(* IEC 61131-3 sources: AXOpen/src/components.cognex.vision/app/src/Documentation, 6 files *)

(* ---- Component_1.st ---- *)
USING AXOpen.Core;

NAMESPACE AXOpen.Components.Cognex.Vision

    {S7.extern=ReadWrite}
    CLASS Component_1 EXTENDS AXOpen.Core.AxoObject
        //<ComponentDeclaration>
        VAR PUBLIC
            Insight_7600 : AXOpen.Components.Cognex.Vision.v_6_0_0_0.AxoInsight;
        END_VAR
        //</ComponentDeclaration>

        //<InitializationArgumentsDeclaration>
        VAR PUBLIC
            {#ix-set:AttributeName = "<#Activate manual control#>"}
            ActivateManualControl : BOOL;
        END_VAR
        //</InitializationArgumentsDeclaration>

        METHOD PUBLIC OVERRIDE Run
            VAR_INPUT
                parent : IAxoObject;
            END_VAR

            SUPER.Run(parent);

            IF ActivateManualControl THEN
                //<InsightManualControl>
                Insight_7600.ActivateManualControl();
                //</InsightManualControl>
            END_IF;

            //<Initialization>
            Insight_7600.Run(parent := THIS, hwID :=  HwIdentifiers#is7600_HwID);
            //</Initialization>
            THIS.UseInSequencer();
        END_METHOD

        //<Usage>
        VAR PUBLIC
            Sequencer : AxoSequencer;
            Steps : ARRAY[0..10] OF AXOpen.Core.AxoStep;
        END_VAR

        VAR PRIVATE
            _InspectionResults  :   AXOpen.Components.Cognex.Vision.v_6_0_0_0.AxoInsight_ResultData;
        END_VAR

        METHOD PRIVATE UseInSequencer
            IF Sequencer.GetContext().OpenCycleCount() <= ULINT#10 THEN
                Sequencer.SequenceMode := eAxoSequenceMode#RunOnce;
            END_IF;

            Sequencer.Run(THIS);
            Sequencer.Open();

            IF(Steps[0].Execute(Sequencer, 'Restore')) THEN
                Insight_7600.Restore();
                Sequencer.MoveNext();
            END_IF;

            IF(Steps[1].Execute(Sequencer, 'Change job: 1_test01.job')) THEN
                IF(Insight_7600.ChangeJob('1_test01.job').IsDone()) THEN
                    Sequencer.MoveNext();
                END_IF;
            END_IF;

            IF(Steps[2].Execute(Sequencer, 'Trigger')) THEN
                IF(Insight_7600.Trigger().IsDone()) THEN
                    Sequencer.MoveNext();
                END_IF;
            END_IF;

            IF(Steps[3].Execute(Sequencer, 'Evaluate inspection results')) THEN
                _InspectionResults := Insight_7600.InspectionResults;
                Sequencer.MoveNext();
            END_IF;

            IF(Steps[4].Execute(Sequencer, 'Clear inspaction results')) THEN
                IF(Insight_7600.ClearInspectionResults().IsDone()) THEN
                    Sequencer.MoveNext();
                END_IF;
            END_IF;

            IF(Steps[5].Execute(Sequencer, 'Soft event')) THEN
                IF(Insight_7600.SoftEvent(UINT#5).IsDone()) THEN
                    Sequencer.MoveNext();
                END_IF;
            END_IF;

            IF(Steps[6].Execute(Sequencer, 'Restore')) THEN
                Insight_7600.Restore();
                Sequencer.CompleteSequence();
            END_IF;

        END_METHOD

        //</Usage>

    END_CLASS
END_NAMESPACE

(* ---- Component_2.st ---- *)
USING AXOpen.Core;

NAMESPACE AXOpen.Components.Cognex.Vision.v_6_0_0_0

    {S7.extern=ReadWrite}
    CLASS Component_2 EXTENDS AXOpen.Core.AxoObject
        //<ComponentDeclaration>
        VAR PUBLIC
            Dataman_280 : AXOpen.Components.Cognex.Vision.v_6_0_0_0.AxoDataman;
        END_VAR
        //</ComponentDeclaration>

        //<InitializationArgumentsDeclaration>
        VAR PUBLIC
            {#ix-set:AttributeName = "<#Activate manual control#>"}
            ActivateManualControl : BOOL;
        END_VAR
        //</InitializationArgumentsDeclaration>

        METHOD PUBLIC OVERRIDE Run
            VAR_INPUT
                parent : IAxoObject;
            END_VAR

            SUPER.Run(parent);

            IF ActivateManualControl THEN
                //<DatamanManualControl>
                Dataman_280.ActivateManualControl();
                //</DatamanManualControl>
            END_IF;

            //<Initialization>
            Dataman_280.Run(parent  :=  THIS, hwID :=  HwIdentifiers#dm_280_HwID);
            //</Initialization>

            THIS.UseInSequencer();
        END_METHOD

        //<Usage>
        VAR PUBLIC
            Sequencer : AxoSequencer;
            Steps : ARRAY[0..10] OF AXOpen.Core.AxoStep;
        END_VAR

        VAR PRIVATE
            _ResultData  :   AXOpen.Components.Cognex.Vision.v_6_0_0_0.AxoDataman_ResultData;
        END_VAR

        METHOD PRIVATE UseInSequencer
            IF Sequencer.GetContext().OpenCycleCount() <= ULINT#10 THEN
                Sequencer.SequenceMode := eAxoSequenceMode#RunOnce;
            END_IF;

            Sequencer.Run(THIS);
            Sequencer.Open();

            IF(Steps[0].Execute(Sequencer, 'Restore')) THEN
                Dataman_280.Restore();
                Sequencer.MoveNext();
            END_IF;

            IF(Steps[1].Execute(Sequencer, 'Clear result data')) THEN
                IF(Dataman_280.ClearResultData().IsDone()) THEN
                    Sequencer.MoveNext();
                END_IF;
            END_IF;

            IF(Steps[2].Execute(Sequencer, 'Read data')) THEN
                IF(Dataman_280.Read().IsDone()) THEN
                    Sequencer.MoveNext();
                END_IF;
            END_IF;

            IF(Steps[3].Execute(Sequencer, 'Evaluate data')) THEN
                _ResultData := Dataman_280.ResultData;
                Sequencer.MoveNext();
            END_IF;

            IF(Steps[4].Execute(Sequencer, 'Restore')) THEN
                Dataman_280.Restore();
                Sequencer.CompleteSequence();
            END_IF;

        END_METHOD

        //</Usage>
    END_CLASS
END_NAMESPACE

(* ---- Component_3.st ---- *)
USING AXOpen.Core;

NAMESPACE AXOpen.Components.Cognex.Vision

    {S7.extern=ReadWrite}
    CLASS Component_3 EXTENDS AXOpen.Core.AxoObject
        //<ComponentDeclaration>
        VAR PUBLIC
            Dataman_300 : AXOpen.Components.Cognex.Vision.v_6_0_0_0.AxoDataman;
        END_VAR
        //</ComponentDeclaration>

        //<InitializationArgumentsDeclaration>
        VAR PUBLIC
            {#ix-set:AttributeName = "<#Activate manual control#>"}
            ActivateManualControl : BOOL;
        END_VAR
        //</InitializationArgumentsDeclaration>

        METHOD PUBLIC OVERRIDE Run
            VAR_INPUT
                parent : IAxoObject;
            END_VAR

            SUPER.Run(parent);

            IF ActivateManualControl THEN
                //<DatamanManualControl>
                Dataman_300.ActivateManualControl();
                //</DatamanManualControl>
            END_IF;

            //<Initialization>
            Dataman_300.Run(parent := THIS, hwID :=  HwIdentifiers#dm_300_HwID);
            //</Initialization>

        THIS.UseInSequencer();
        END_METHOD

        //<Usage>
        VAR PUBLIC
            Sequencer : AxoSequencer;
            Steps : ARRAY[0..10] OF AXOpen.Core.AxoStep;
        END_VAR

        VAR PRIVATE
            _ResultData  :   AXOpen.Components.Cognex.Vision.v_6_0_0_0.AxoDataman_ResultData;
        END_VAR

        METHOD PRIVATE UseInSequencer
            IF Sequencer.GetContext().OpenCycleCount() <= ULINT#10 THEN
                Sequencer.SequenceMode := eAxoSequenceMode#RunOnce;
            END_IF;

            Sequencer.Run(THIS);
            Sequencer.Open();

            IF(Steps[0].Execute(Sequencer, 'Restore')) THEN
                Dataman_300.Restore();
                Sequencer.MoveNext();
            END_IF;

            IF(Steps[1].Execute(Sequencer, 'Clear result data')) THEN
                IF(Dataman_300.ClearResultData().IsDone()) THEN
                    Sequencer.MoveNext();
                END_IF;
            END_IF;

            IF(Steps[2].Execute(Sequencer, 'Read data')) THEN
                IF(Dataman_300.Read().IsDone()) THEN
                    Sequencer.MoveNext();
                END_IF;
            END_IF;

            IF(Steps[3].Execute(Sequencer, 'Evaluate data')) THEN
                _ResultData := Dataman_300.ResultData;
                Sequencer.MoveNext();
            END_IF;

            IF(Steps[4].Execute(Sequencer, 'Restore')) THEN
                Dataman_300.Restore();
                Sequencer.CompleteSequence();
            END_IF;

        END_METHOD

        //</Usage>
    END_CLASS
END_NAMESPACE

(* ---- Component_4.st ---- *)
USING AXOpen.Core;

NAMESPACE AXOpen.Components.Cognex.Vision

    {S7.extern=ReadWrite}
    CLASS Component_4 EXTENDS AXOpen.Core.AxoObject
        //<ComponentDeclaration>
        VAR PUBLIC
            Insight_2800 : AXOpen.Components.Cognex.Vision.v_24_0_0.AxoInsight;
        END_VAR
        //</ComponentDeclaration>

        //<InitializationArgumentsDeclaration>
        VAR PUBLIC
            {#ix-set:AttributeName = "<#Activate manual control#>"}
            ActivateManualControl : BOOL;
        END_VAR
        //</InitializationArgumentsDeclaration>

        METHOD PUBLIC OVERRIDE Run
            VAR_INPUT
                inParent : IAxoObject;
            END_VAR

            SUPER.Run(inParent);

            IF ActivateManualControl THEN
                //<InsightManualControl>
                Insight_2800.ActivateManualControl();
                //</InsightManualControl>
            END_IF;

            //<Initialization>
            Insight_2800.Run(parent := THIS, hwID := HwIdentifiers#is2800_HwID);
            //</Initialization>
            THIS.UseInSequencer();
        END_METHOD

        //<Usage>
        VAR PUBLIC
            Sequencer : AxoSequencer;
            Steps : ARRAY[0..14] OF AXOpen.Core.AxoStep;
        END_VAR

        VAR PRIVATE
            _InspectionResults  :   AXOpen.Components.Cognex.Vision.v_24_0_0.AxoInsight_ResultData;
            _UserData           :   AXOpen.Components.Cognex.Vision.v_24_0_0.AxoInsight_UserData;
        END_VAR

        METHOD PRIVATE UseInSequencer
            IF Sequencer.GetContext().OpenCycleCount() <= ULINT#10 THEN
                Sequencer.SequenceMode := eAxoSequenceMode#RunOnce;
            END_IF;

            Sequencer.Run(THIS);
            Sequencer.Open();

            IF(Steps[0].Execute(Sequencer, 'Restore')) THEN
                Insight_2800.Restore();
                Sequencer.MoveNext();
            END_IF;

            IF(Steps[1].Execute(Sequencer, 'Change job by number:2')) THEN
                IF(Insight_2800.ChangeJob(UINT#2).IsDone()) THEN
                    Sequencer.MoveNext();
                END_IF;
            END_IF;

            IF(Steps[2].Execute(Sequencer, 'Change job by name:1_BOGE_Lavy_pedal_090_091')) THEN
                IF(Insight_2800.ChangeJob('1_BOGE_Lavy_pedal_090_091').IsDone()) THEN
                    Sequencer.MoveNext();
                END_IF;
            END_IF;

            IF(Steps[3].Execute(Sequencer, 'Trigger')) THEN
                IF(Insight_2800.Trigger().IsDone()) THEN
                    Sequencer.MoveNext();
                END_IF;
            END_IF;

            IF(Steps[4].Execute(Sequencer, 'Evaluate inspection results')) THEN
                _InspectionResults := Insight_2800.InspectionResults;
                Sequencer.MoveNext();
            END_IF;

            IF(Steps[5].Execute(Sequencer, 'Clear inspection results')) THEN
                IF(Insight_2800.ClearInspectionResults().IsDone()) THEN
                    Sequencer.MoveNext();
                END_IF;
            END_IF;

            IF(Steps[6].Execute(Sequencer, 'Soft event:5')) THEN
                IF(Insight_2800.SoftEvent(UINT#5).IsDone()) THEN
                    Sequencer.MoveNext();
                END_IF;
            END_IF;

            IF(Steps[7].Execute(Sequencer, 'Clear user data')) THEN
                IF(Insight_2800.ClearUserData().IsDone()) THEN
                    Sequencer.MoveNext();
                END_IF;
            END_IF;

            IF(Steps[8].Execute(Sequencer, 'Set user data as byte')) THEN
                IF(Insight_2800.SetUserDataAsByte(BYTE#12,UINT#0)) THEN
                    Sequencer.MoveNext();
                END_IF;
            END_IF;

            IF(Steps[9].Execute(Sequencer, 'Set user data as string')) THEN
                IF(Insight_2800.SetUserDataAsString('Set user data string l24',UINT#1)) THEN
                    Sequencer.MoveNext();
                END_IF;
            END_IF;

            IF(Steps[10].Execute(Sequencer, 'Set user data as dint')) THEN
                IF(Insight_2800.SetUserDataAsDint(DINT#123456,UINT#25)) THEN
                    Sequencer.MoveNext();
                END_IF;
            END_IF;

            IF(Steps[11].Execute(Sequencer, 'Set user data as real')) THEN
                IF(Insight_2800.SetUserDataAsReal(REAL#789.123,UINT#29)) THEN
                    Sequencer.MoveNext();
                END_IF;
            END_IF;

            IF(Steps[12].Execute(Sequencer, 'Send already prepared user data')) THEN
                IF(Insight_2800.SendUserData().IsDone()) THEN
                    Sequencer.MoveNext();
                END_IF;
            END_IF;

            IF(Steps[13].Execute(Sequencer, 'Send user data passed as input variable')) THEN
                _UserData.Data[0] := BYTE#65;
                // ..
                // ..
                _UserData.Data[27] := BYTE#32;

                IF(Insight_2800.SendUserData(_UserData, UINT#32).IsDone()) THEN
                    Sequencer.MoveNext();
                END_IF;
            END_IF;

            IF(Steps[14].Execute(Sequencer, 'Restore')) THEN
                Insight_2800.Restore();
                Sequencer.CompleteSequence();
            END_IF;
        END_METHOD

        //</Usage>

    END_CLASS
END_NAMESPACE

(* ---- Component_5.st ---- *)
USING AXOpen.Core;

NAMESPACE AXOpen.Components.Cognex.Vision

    {S7.extern=ReadWrite}
    CLASS Component_5 EXTENDS AXOpen.Core.AxoObject
        //<ComponentDeclaration>
        VAR PUBLIC
            VisionPro : AXOpen.Components.Cognex.Vision.AxoVisionPro;
        END_VAR
        //</ComponentDeclaration>

        //<InitializationArgumentsDeclaration>
        VAR PUBLIC
            {#ix-set:AttributeName = "<#Activate manual control#>"}
            ActivateManualControl : BOOL;
        END_VAR
        //</InitializationArgumentsDeclaration>

        METHOD PUBLIC OVERRIDE Run
            VAR_INPUT
                parent : IAxoObject;
            END_VAR

            SUPER.Run(parent);

            IF ActivateManualControl THEN
                //<InsightManualControl>
                VisionPro.ActivateManualControl();
                //</InsightManualControl>
            END_IF;

            //<Initialization>
            // VisionPro.Run(parent := THIS, hwID := HwIdentifiers#vision_pro_HwID, CameraNo := BYTE#1);
            VisionPro.Run(parent := THIS, hwID := HwIdentifiers#CommunicationCard_HwID, CameraNo := BYTE#1);
            //</Initialization>
            THIS.UseInSequencer();
        END_METHOD

        //<Usage>
        VAR PUBLIC
            Sequencer : AxoSequencer;
            Steps : ARRAY[0..10] OF AXOpen.Core.AxoStep;
        END_VAR

        VAR PRIVATE
            _InspectionResults : ARRAY[0..1300] OF BYTE;
            _UserData : ARRAY[0..1300] OF BYTE;
        END_VAR

        METHOD PRIVATE UseInSequencer
            IF Sequencer.GetContext().OpenCycleCount() <= ULINT#10 THEN
                Sequencer.SequenceMode := eAxoSequenceMode#RunOnce;
            END_IF;

            Sequencer.Run(THIS);
            Sequencer.Open();

            IF(Steps[0].Execute(Sequencer, 'Restore')) THEN
                VisionPro.Restore();
                Sequencer.MoveNext();
            END_IF;

            IF(Steps[1].Execute(Sequencer, 'HardResetAllCameras')) THEN
                IF(VisionPro.HardResetAllCameras().IsDone()) THEN
                    Sequencer.MoveNext();
                END_IF;
            END_IF;

            IF(Steps[2].Execute(Sequencer, 'SendData')) THEN
                IF(VisionPro.SendData(InspectionType := BYTE#1, BufferID := BYTE#0, JobID := BYTE#1, Length := UINT#1, Data := _UserData).IsDone()) THEN
                    Sequencer.MoveNext();
                END_IF;
            END_IF;

            IF(Steps[3].Execute(Sequencer, 'Trigger')) THEN
                IF(VisionPro.Trigger().IsDone()) THEN
                    Sequencer.MoveNext();
                END_IF;
            END_IF;

            IF(Steps[4].Execute(Sequencer, 'SendData')) THEN
                IF(VisionPro.SendData(InspectionType := BYTE#2, BufferID := BYTE#0, JobID := BYTE#1, Length := UINT#1, Data := _UserData).IsDone()) THEN
                    Sequencer.MoveNext();
                END_IF;
            END_IF;

            IF(Steps[5].Execute(Sequencer, 'ReadResults')) THEN
                IF(VisionPro.ReadResults(JobID := BYTE#1, Length := UINT#620, Data := _InspectionResults).IsDone()) THEN
                    Sequencer.MoveNext();
                END_IF;
            END_IF;

            IF(Steps[6].Execute(Sequencer, 'Reset')) THEN
                IF(VisionPro.Reset().IsDone()) THEN
                    Sequencer.MoveNext();
                END_IF;
            END_IF;

            IF(Steps[7].Execute(Sequencer, 'Restore')) THEN
                VisionPro.Restore();
                Sequencer.CompleteSequence();
            END_IF;
        END_METHOD

        //</Usage>

    END_CLASS
END_NAMESPACE

(* ---- DocumentationContext.st ---- *)
NAMESPACE AXOpen.Components.Cognex.Vision.v_6_0_0_0

    {S7.extern=ReadWrite}
    CLASS DocumentationContext EXTENDS AXOpen.Core.AxoContext
        VAR PUBLIC
            _rootObject :   AxoObject;
            componentOne : Component_1;
            componentTwo : Component_2;
            componentThree : Component_3;
        END_VAR

        METHOD PROTECTED OVERRIDE Main
            THIS.InitializeRootObject(_rootObject);
            componentOne.Run(_rootObject);
            componentTwo.Run(_rootObject);
            componentThree.Run(_rootObject);
        END_METHOD
    END_CLASS
END_NAMESPACE
